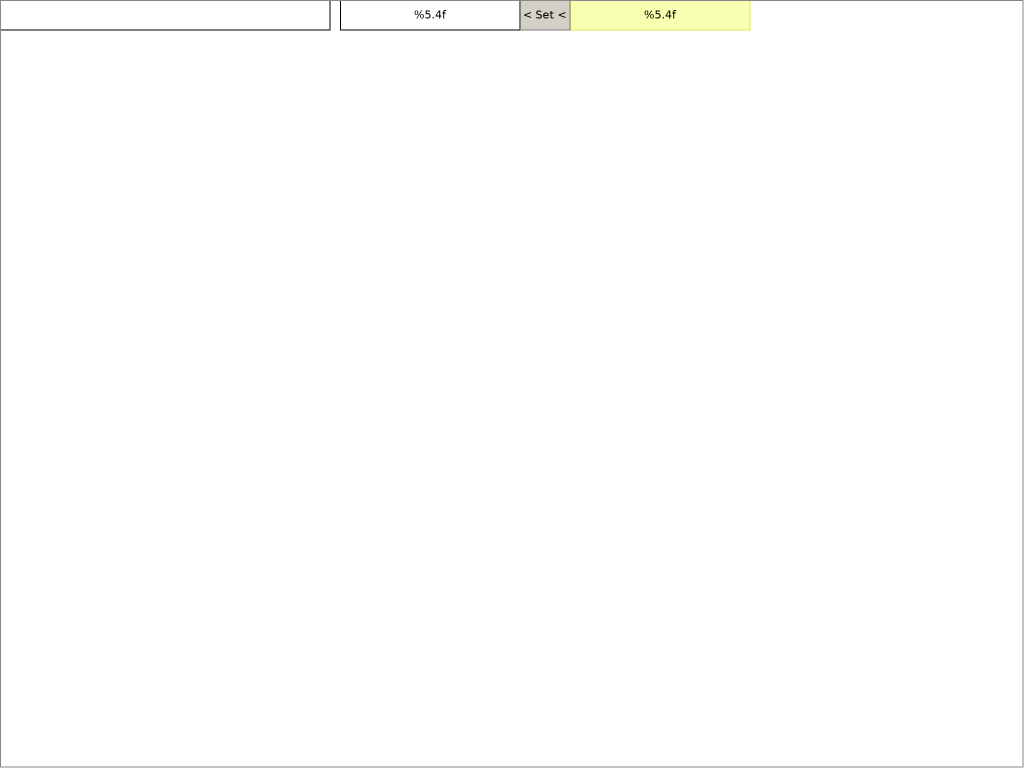
VISUALIZATION Param_LREAL_Pparam  // 1024x768
VAR_INPUT
	nIdx:		INT;
END_VAR
    Rectangle (340,0 180x30), "%5.4f", text variable: stPParam_Visu.fLrealAktValue[nIdx]
    Rectangle (0,0 330x30), text list: 'TL_Pparmas', text index: nIdx
    Rectangle (570,0 180x30), "%5.4f", text variable: stPParam_Visu.fLrealNewValue[nIdx]
        OnMouseClick: write the text variable via Default
    Rectangle (520,0 50x30), "< Set <"
        OnMouseClick: execute { stPParam_Visu.bLrealSetValue[nIdx]:=TRUE; }
END_VISUALIZATION

(* stored: Version 1.1.0.1, ProductVersion 3.1.4024.12
   Visu Param_LREAL_Pparam: Id {637fe378-de00-4a80-b17a-6f07a54d2b24} *)
